// TIA Portal V18 export
FUNCTION_BLOCK "НулевыеБлокировки"   // FB39, FBD
{ S7_Optimized_Access := 'TRUE' }
VERSION : 0.1
// stored: AutoNumber true, IsIECCheckEnabled false, IsRetainMemResEnabled false, MemoryReserve 100, SetENOAutomatically false, UDAEnableTagReadback false
   VAR_INPUT
      x_Nok : Bool;
   END_VAR
   VAR_OUTPUT
      y_ERROR : Bool := true;
   END_VAR
   VAR_IN_OUT
      ton_delay : Time := T#1s;
   END_VAR
   VAR
      IEC_Timer_0_Instance { S7_SetPoint := 'True'} : TON_TIME;
   END_VAR
   VAR_TEMP
      ton_elapsed : Bool;
   END_VAR
BEGIN

REGION Network 1
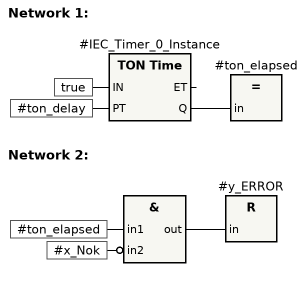
   #IEC_Timer_0_Instance(IN := true, PT := #ton_delay);   // TON
   #ton_elapsed := #IEC_Timer_0_Instance.Q;
END_REGION

REGION Network 2
   IF #ton_elapsed AND NOT #x_Nok THEN #y_ERROR := FALSE; END_IF;
END_REGION
END_FUNCTION_BLOCK
